{attribute addProperty BoxType "EL5101-0000-1019"}
{attribute addProperty Id "ENC_Status_compactAT %I*ENC_Status_compact_A61A67D1160200ENC_Control_compactAT %Q*ENC_Control_compact_ADEB38374860WcStateAT %I*WcState_98A4DF7520.250InfoDataAT %I*InfoData_BC63D37F80100"}
{attribute addProperty CRC "1201638637"}
{attribute addProperty SizeInBites "290"}
{attribute addProperty SizeInBytes "36.25"}
TYPE EL5101_2133D810 :
STRUCT
	{attribute addProperty Name "ENC_Status_compact"}
	ENC_Status_compact : ENC_Status_compact_A61A67D1;
	{attribute addProperty Name "ENC_Control_compact"}
	ENC_Control_compact : ENC_Control_compact_ADEB3837;
	{attribute addProperty Name "WcState"}
	WcState : WcState_98A4DF75;
	{attribute addProperty Name "InfoData"}
	InfoData : InfoData_BC63D37F;
END_STRUCT
END_TYPE

(* stored: Version 1.2.0.0, ProductVersion 3.1.4024.9
   DUT EL5101_2133D810: Id {034962ab-cd08-4de6-9f5e-a2280d8a1148} *)
